TYPE U_Chamber1_ServiceCtrlView :
UNION
	ByName : ST_Chamber1_ServiceCtrl;
	ByIndex : ARRAY[1..GVL_Chamber1_Config.cServiceCount] OF ST_ServiceCtrl;
END_UNION
END_TYPE

(* stored: Version 1.1.0.1, ProductVersion 3.1.4026.18
   DUT U_Chamber1_ServiceCtrlView: Id {ebffcb9a-149a-4b8d-9ee4-49df4adc4fb1} *)
